FUNCTION_BLOCK FB_Observer_DINT EXTENDS FB_AbstractObserver
VAR
    _nVal:              DINT;
END_VAR

METHOD FB_init : BOOL
VAR_INPUT
	bInitRetains : BOOL; // if TRUE, the retain variables are initialized (warm start / cold start)
	bInCopyCode : BOOL;  // if TRUE, the instance afterwards gets moved into the copy code (online change)
END_VAR
THIS^._nTypeClass := __SYSTEM.TYPE_CLASS.TYPE_DINT;
THIS^._pVal := ADR(THIS^._nVal);
THIS^._nSize := SIZEOF(THIS^._nVal);
END_METHOD

PROPERTY nValue32 : DINT
GET
nValue32 := THIS^._nVal;
END_GET
END_PROPERTY

END_FUNCTION_BLOCK

(* stored: Version 1.1.0.1, ProductVersion 3.1.4024.12
   POU FB_Observer_DINT: Id {22c8b8ae-99d5-4d37-9e7c-afe4e3df0815}, SpecialFunc None
   Method FB_init: Id {57d61c6e-d332-0a6d-2a04-53728b26bdc9}
   Property nValue32: Id {bec0dc45-8824-4d58-907b-b755df6d4f5b}
   Get Get: Id {1c41b536-f2de-4d2e-a865-45917af5498b} *)
